{attribute 'linkalways'} 
{attribute 'no_explicit_call' := 'This FB is a CLASS and must be accessed using methods or properties'}
{attribute 'enable_dynamic_creation'}
FUNCTION_BLOCK Node_F_VN_SetAt_TcVnVector4_SINT EXTENDS VisionNode
VAR
    aElement : _TcVnVector4_SINT;
    ipContainer : _ITcVnContainer;
    nIndex : _ULINT(0);
    hrPrev : _HRESULT(S_OK);
    hresult : _HRESULT(S_OK);
END_VAR

METHOD PUBLIC  Clone : I_Node
VAR
	pNode : POINTER TO Node_F_VN_SetAt_TcVnVector4_SINT;
END_VAR
pNode := __NEW(Node_F_VN_SetAt_TcVnVector4_SINT);
Clone := pNode^;
END_METHOD

METHOD FB_init : BOOL
VAR_INPUT
	bInitRetains : BOOL; // if TRUE, the retain variables are initialized (warm start / cold start)
	bInCopyCode : BOOL;  // if TRUE, the instance afterwards gets moved into the copy code (online change)
END_VAR
AddInput('aElement', aElement);
AddInput('ipContainer', ipContainer);
AddInput('nIndex', nIndex);
AddInput('hrPrev', hrPrev);
AddOutput('ipContainer', ipContainer);
AddOutput('hresult',hresult);
END_METHOD

METHOD PROTECTED OnExecute : HRESULT
hresult.Value := F_VN_SetAt_TcVnVector4_SINT(
    aElement := aElement.Value,
    ipContainer := ipContainer.Value,
    nIndex := nIndex.Value,
    hrPrev:= hrPrev.Value);
END_METHOD

METHOD PUBLIC PreExecutionCheck
VAR_INPUT
	Check : I_PreExecutionChecks;
END_VAR
Check.IsTrue(ipContainer.IsValid, 'ipContainer must be a valid container');
END_METHOD

END_FUNCTION_BLOCK

(* stored: Version 1.1.0.1, ProductVersion 3.1.4024.13
   POU Node_F_VN_SetAt_TcVnVector4_SINT: Id {0a2cf473-e454-4e4e-8fa3-726e11023731}, SpecialFunc None
   Folder Constructor: Id {1e88f81a-7293-4414-a011-345e0197b8c5}
   Method Clone: Id {08059807-b63c-4065-9461-f68ed34a40f1}
   Method FB_init: Id {3256cf06-a22c-41a5-8888-7a6ee9fdd833}
   Method OnExecute: Id {a481b3ed-a40e-4c1b-807e-0e6ea07f235d}
   Method PreExecutionCheck: Id {a262d539-a403-44bd-9865-9d3dd397b7db} *)
